(* IEC 61131-3 sources: AXOpen/src/components.rexroth.press/app/SystemConstants, 2 files *)

(* ---- plc_line_IoAddresses.st ---- *)
CONFIGURATION IoAddresses
    VAR_GLOBAL

        // Module rexroth_press/Input_24_Words
        rexroth_press_Input_24_Words_Input AT %IB0 : rexroth_press_Input_24_Words_Input_Layout;

        // Module rexroth_press/Output_21_Words
        rexroth_press_Output_21_Words_Output AT %QB0 : rexroth_press_Output_21_Words_Output_Layout;

        // Module rexroth_press/ParamCh_5Words
        rexroth_press_ParamCh_5Words_Input AT %IB48 : rexroth_press_ParamCh_5Words_Input_Layout;
        rexroth_press_ParamCh_5Words_Output AT %QB42 : rexroth_press_ParamCh_5Words_Output_Layout;
    END_VAR
END_CONFIGURATION

TYPE
    rexroth_press_Input_24_Words_Input_Layout : STRUCT
        Signals_0 AT %B0 : WORD;
        Signals_1 AT %B2 : WORD;
        Signals_2 AT %B4 : WORD;
        Signals_3 AT %B6 : WORD;
        Signals_4 AT %B8 : WORD;
        Signals_5 AT %B10 : WORD;
        Signals_6 AT %B12 : WORD;
        Signals_7 AT %B14 : WORD;
        Signals_8 AT %B16 : WORD;
        Signals_9 AT %B18 : WORD;
        Signals_10 AT %B20 : WORD;
        Signals_11 AT %B22 : WORD;
        Signals_12 AT %B24 : WORD;
        Signals_13 AT %B26 : WORD;
        Signals_14 AT %B28 : WORD;
        Signals_15 AT %B30 : WORD;
        Signals_16 AT %B32 : WORD;
        Signals_17 AT %B34 : WORD;
        Signals_18 AT %B36 : WORD;
        Signals_19 AT %B38 : WORD;
        Signals_20 AT %B40 : WORD;
        Signals_21 AT %B42 : WORD;
        Signals_22 AT %B44 : WORD;
        Signals_23 AT %B46 : WORD;
    END_STRUCT;
END_TYPE

TYPE
    rexroth_press_Output_21_Words_Output_Layout : STRUCT
        Signals_0 AT %B0 : WORD;
        Signals_1 AT %B2 : WORD;
        Signals_2 AT %B4 : WORD;
        Signals_3 AT %B6 : WORD;
        Signals_4 AT %B8 : WORD;
        Signals_5 AT %B10 : WORD;
        Signals_6 AT %B12 : WORD;
        Signals_7 AT %B14 : WORD;
        Signals_8 AT %B16 : WORD;
        Signals_9 AT %B18 : WORD;
        Signals_10 AT %B20 : WORD;
        Signals_11 AT %B22 : WORD;
        Signals_12 AT %B24 : WORD;
        Signals_13 AT %B26 : WORD;
        Signals_14 AT %B28 : WORD;
        Signals_15 AT %B30 : WORD;
        Signals_16 AT %B32 : WORD;
        Signals_17 AT %B34 : WORD;
        Signals_18 AT %B36 : WORD;
        Signals_19 AT %B38 : WORD;
        Signals_20 AT %B40 : WORD;
    END_STRUCT;
END_TYPE

TYPE
    rexroth_press_ParamCh_5Words_Input_Layout : STRUCT
        Signals_0 AT %B0 : WORD;
        Signals_1 AT %B2 : WORD;
        Signals_2 AT %B4 : WORD;
        Signals_3 AT %B6 : WORD;
        Signals_4 AT %B8 : WORD;
    END_STRUCT;
END_TYPE

TYPE
    rexroth_press_ParamCh_5Words_Output_Layout : STRUCT
        Signals_5 AT %B0 : WORD;
        Signals_6 AT %B2 : WORD;
        Signals_7 AT %B4 : WORD;
        Signals_8 AT %B6 : WORD;
        Signals_9 AT %B8 : WORD;
    END_STRUCT;
END_TYPE

(* ---- plc_line_HwIdentifiers.st ---- *)
CONFIGURATION HardwareIDs
    VAR_GLOBAL CONSTANT
        plc_line_HwID : UINT := UINT#32;
        plc_line_Rail_0_HwID : UINT := UINT#268;
        plc_line_plc_line_HwID : UINT := UINT#48;
        plc_line_plc_line_CPU_display_1_HwID : UINT := UINT#54;
        plc_line_plc_line_Card_reader_writer_1_HwID : UINT := UINT#51;
        plc_line_plc_line_DP_interface_1_HwID : UINT := UINT#60;
        plc_line_plc_line_OPC_UA_1_HwID : UINT := UINT#117;
        plc_line_plc_line_PROFINET_interface_1_HwID : UINT := UINT#64;
        plc_line_plc_line_PROFINET_interface_1_Port_1_HwID : UINT := UINT#65;
        plc_line_plc_line_PROFINET_interface_1_Port_2_HwID : UINT := UINT#66;
        plc_line_plc_line_PROFINET_interface_2_HwID : UINT := UINT#72;
        plc_line_plc_line_PROFINET_interface_2_Port_3_HwID : UINT := UINT#73;
        plc_line_plc_line_Virtual_communication_interface_HwID : UINT := UINT#135;
        profinet_plc_line_HwID : UINT := UINT#256;
        rexroth_press_HwID : UINT := UINT#258;
        rexroth_press_F_Modul_not_used_ID_FMod_NotUsed_HwID : UINT := UINT#266;
        rexroth_press_Input_24_Words_ID_InMod_24Words_HwID : UINT := UINT#264;
        rexroth_press_Output_21_Words_ID_OutMod_21Words_HwID : UINT := UINT#263;
        rexroth_press_ParamCh_5Words_ID_PaCh_5Words_HwID : UINT := UINT#265;
        rexroth_press_Rack_HwID : UINT := UINT#261;
        rexroth_press_rexroth_press_HwID : UINT := UINT#262;
        rexroth_press_rexroth_press_DAP_1_HwID : UINT := UINT#267;
        rexroth_press_rexroth_press_PN_IO_HwID : UINT := UINT#257;
        rexroth_press_rexroth_press_PN_IO_Port_1_HwID : UINT := UINT#259;
        rexroth_press_rexroth_press_PN_IO_Port_2_HwID : UINT := UINT#260;

    END_VAR
END_CONFIGURATION
